Staubli VAL3: findInWhichBox1.pgx

program findInWhichBox1(string& x_sLodaBox1[])
  local num i
  local num l_nResult
  local point l_pHere
  local tool l_tTool
  local num j
  local num k
  local num l_nAngle
  local num l_nPointIndex
  local num m
  local num l_nShort
  local bool l_bCondition
  local num l_nSize
begin

  //分析比较最可能的安全盒子
  l_nSize=size(nInWhichBox)
  resize(nShortP2PAngle,1,l_nSize)
  resize(nShortP2PDists,1,l_nSize)
  for k=0 to size(nShortP2PDists)-1
    nShortP2PAngle[k]=9999
    nShortP2PDists[k]=9999
  endFor
  for i=0 to size(nInWhichBox)-1


      call getTrajTool(l_tTool,sml:box[sBox1[i]].nIndexGun )
      l_pHere=here(l_tTool,world)
      l_bCondition=false
      for j=0 to size(sml:box[sBox1[i]].comment)-1
        if left(sml:box[sBox1[i]].comment[j],1)=="#"
          call _getP2PAngle(l_pHere,sml:box[sBox1[i]].pPointRx[j],l_nAngle)
          if nShortP2PAngle[i]>l_nAngle and l_nAngle<=15
            nShortP2PAngle[i]=l_nAngle
            l_bCondition=true
            l_nPointIndex=j
          endIf
        endIf
      endFor
      if l_bCondition
        call _getP2PDistance(sml:box[sBox1[i]].pPointRx[l_nPointIndex],l_pHere,nShortP2PDists[i])
      endIf

  endFor
  l_nShort=99999
  for m=0 to size(nShortP2PDists)-1
    if nShortP2PDists[m]<l_nShort
      l_nShort=nShortP2PDists[m]
      x_sLodaBox1=sBox1[nInWhichBox[m]]
    endIf

  endFor
end
